PROGRAM Rep_BE
VAR
	FB_B1520_Rep_Be	:FB_Rep_Ethercat_MURR;
END_VAR

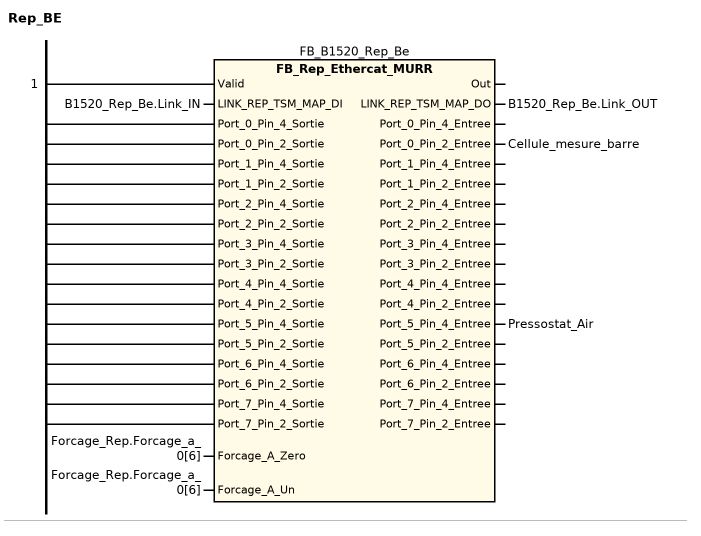
// NETWORK 1
FB_B1520_Rep_Be(
    Valid := TRUE,
    LINK_REP_TSM_MAP_DI := B1520_Rep_Be.Link_IN,
    Port_0_Pin_4_Sortie := TRUE,
    Port_0_Pin_2_Sortie := TRUE,
    Port_1_Pin_4_Sortie := TRUE,
    Port_1_Pin_2_Sortie := TRUE,
    Port_2_Pin_4_Sortie := TRUE,
    Port_2_Pin_2_Sortie := TRUE,
    Port_3_Pin_4_Sortie := TRUE,
    Port_3_Pin_2_Sortie := TRUE,
    Port_4_Pin_4_Sortie := TRUE,
    Port_4_Pin_2_Sortie := TRUE,
    Port_5_Pin_4_Sortie := TRUE,
    Port_5_Pin_2_Sortie := TRUE,
    Port_6_Pin_4_Sortie := TRUE,
    Port_6_Pin_2_Sortie := TRUE,
    Port_7_Pin_4_Sortie := TRUE,
    Port_7_Pin_2_Sortie := TRUE,
    Forcage_A_Zero := Forcage_Rep.Forcage_a_0[6],
    Forcage_A_Un := Forcage_Rep.Forcage_a_0[6],
    LINK_REP_TSM_MAP_DO => B1520_Rep_Be.Link_OUT,
    Port_0_Pin_2_Entree => Cellule_mesure_barre,
    Port_5_Pin_4_Entree => Pressostat_Air); // FB_Rep_Ethercat_MURR

END_PROGRAM

(* stored: Version 1.1.0.1
   POU Rep_BE: Id {b3b1ba5e-e456-4111-8952-9fa38c84c1a2}, SpecialFunc None *)
